{attribute 'qualified_only'}
{attribute 'strict'}
TYPE CoreDriveState :
(
	Init,
	Drive,
	operational,
	stop,
	error,
	BumperStop
);
END_TYPE

(* stored: Version 1.1.0.1, ProductVersion 3.1.4024.11
   DUT CoreDriveState: Id {c2348a90-a5c6-48d0-b159-571f22e67001} *)
